{attribute 'qualified_only'}
{attribute 'strict'}
TYPE eState :
(
	Unconfigured := 0,
	Inactive := 1,
	Active := 2,
	Finalized := 3,
	Configuring := 4,
	CleaningUp := 5,
	Activating := 6,
	Deactivating := 7,
	ShuttingDown := 8,
	ErrorProcessing := 9
);
END_TYPE

(* stored: Version 1.1.0.1, ProductVersion 3.1.4026.18
   DUT eState: Id {a1b2c3d4-1111-1111-1111-111111111111} *)
